// Mitsubishi GX Works2 project: study   PLC: FX3U/FX3UC

PROGRAM MAIN
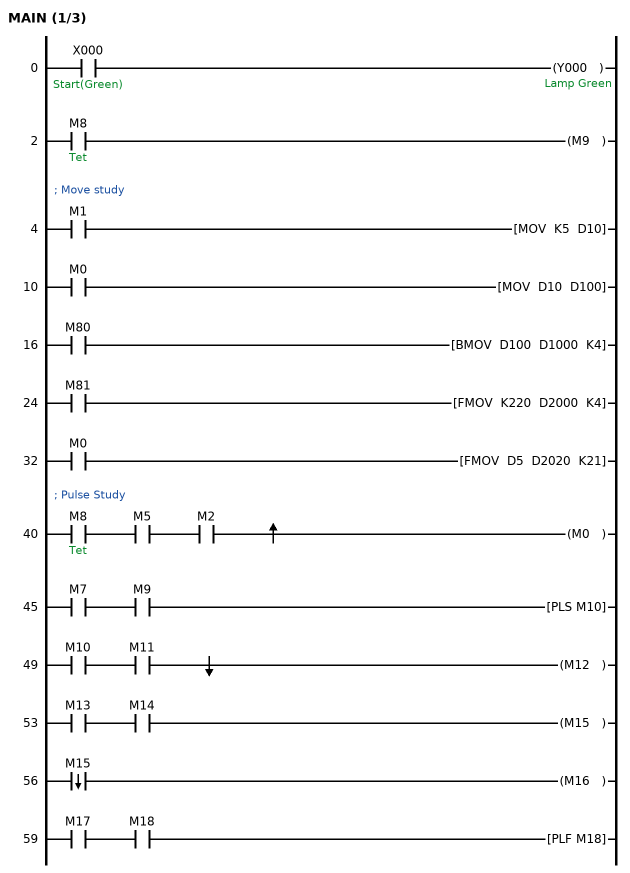
0     LD      X000  ; Start(Green)
      OUT     Y000  ; Lamp Green
2     LD      M8  ; Tet
      OUT     M9
; Move study
4     LD      M1
      MOV     K5 D10
10    LD      M0
      MOV     D10 D100
16    LD      M80
      BMOV    D100 D1000 K4
24    LD      M81
      FMOV    K220 D2000 K4
32    LD      M0
      FMOV    D5 D2020 K21
; Pulse Study
40    LD      M8  ; Tet
      AND     M5
      AND     M2
      MEP
      OUT     M0
45    LD      M7
      AND     M9
      PLS     M10
49    LD      M10
      AND     M11
      MEF
      OUT     M12
53    LD      M13
      AND     M14
      OUT     M15
56    LDF     M15
      OUT     M16
59    LD      M17
      AND     M18
      PLF     M18
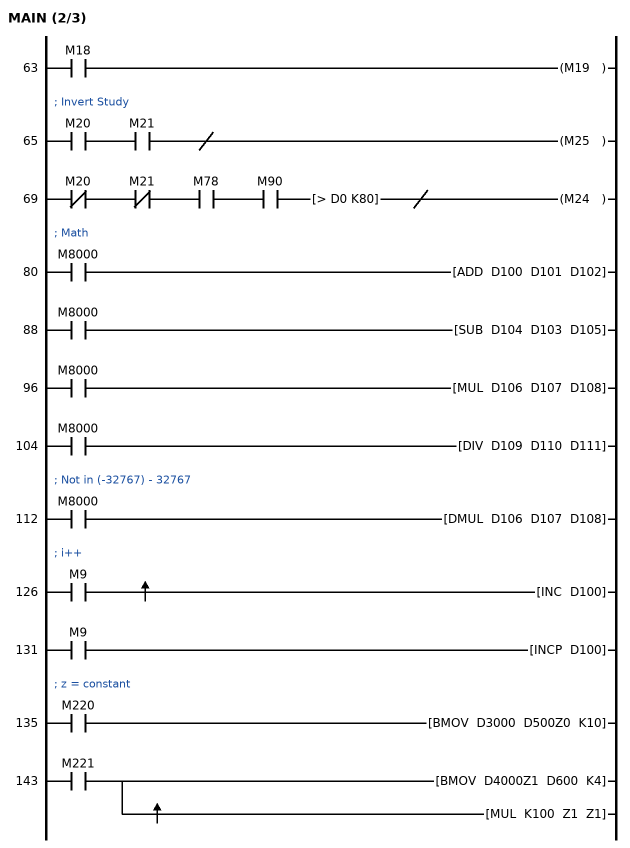
63    LD      M18
      OUT     M19
; Invert Study
65    LD      M20
      AND     M21
      INV
      OUT     M25
69    LDI     M20
      ANI     M21
      AND     M78
      AND     M90
      AND>    D0 K80
      INV
      OUT     M24
; Math
80    LD      M8000
      ADD     D100 D101 D102
88    LD      M8000
      SUB     D104 D103 D105
96    LD      M8000
      MUL     D106 D107 D108
104   LD      M8000
      DIV     D109 D110 D111
; Not in (-32767) - 32767
112   LD      M8000
      DMUL    D106 D107 D108
; i++
126   LD      M9
      MEP
      INC     D100
131   LD      M9
      INCP    D100
; z = constant
135   LD      M220
      BMOV    D3000 D500Z0 K10
143   LD      M221
      BMOV    D4000Z1 D600 K4
      MEP
      MUL     K100 Z1 Z1
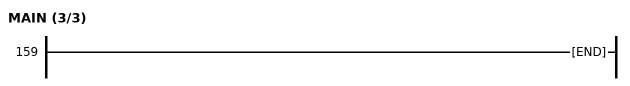
159   END
END_PROGRAM

// device comments not shown above
X001  ; Reset(Yellow)
X002  ; Stop(Red)
X003  ; Sensor1(Camera)
X004  ; Sensor2(Pusher)
Y001  ; Lamp Yellow
Y002  ; Lamp Red
Y003  ; Conveiyor ON
Y005  ; Pusher ON
Y014  ; Camera ON
